// TIA Portal V19 export
TYPE "typeDataFromSafety"
// Safety status
// stored: Access Published, IsFailsafeCompliant true, Namespace Safety
   STRUCT
      safetyReleasedAllSafetyZones { ExternalWritable := 'False'} : Bool;   // All safety zones are released
      ackRequiredAnySafetyZone { ExternalWritable := 'False'} : Bool;   // At least one safety zone requires an acknowledge
      ackOP_changeRequired { ExternalWritable := 'False'} : Bool;   // ACK_OP is waiting for value change
      devicesSummary { ExternalWritable := 'False'} : "Safety.typeDevicesStatusSummary";
      eStopButton0pressed { ExternalWritable := 'False'} : Bool;   // Global - E-stop button E0 is pressed
      eStopButton1pressed { ExternalWritable := 'False'} : Bool;   // Zone 1 - E-stop button E1 is pressed
      fDoor1Open { ExternalWritable := 'False'} : Bool;   // Zone 1 - F-door is open
      AOPD1interrupted { ExternalWritable := 'False'} : Bool;   // Zone 1 - Light curtain is interrupted
      eStopZone1 { ExternalWritable := 'False'} : "Safety.typeEstopFunction";
      fDoorZone1 { ExternalWritable := 'False'} : "Safety.typeFDoorFunction";
      lightCurtainZone1 { ExternalWritable := 'False'} : "Safety.typeAOPD_Function";
      statusZone1 { ExternalWritable := 'False'} : "Safety.typeSafetyZoneStatus";
      activeSTO_Zone1 { ExternalWritable := 'False'} : Bool;   // Zone 1 - STO active
      drive1 { ExternalWritable := 'False'} : "Safety.typeSafetyDrive";
      drive2 { ExternalWritable := 'False'} : "Safety.typeSafetyDrive";
   END_STRUCT;
END_TYPE
